PROGRAM PRG_Process
VAR
	iTank : INT ;
END_VAR




iTank := iTank + 1 ;

END_PROGRAM

(* stored: Version 1.1.0.1, ProductVersion 3.1.4024.12
   POU PRG_Process: Id {80ae12b7-815f-4bcb-8300-fa0ba320e943}, SpecialFunc None *)
